(* PLC project SafeLOGIC, BrAutomation SafeDESIGNER  5.24.1.0 *)
(* stored: companyURL http://www.br-automation.com, creationDateTime Fri Nov 28 14:27:25 2025 *)

PROGRAM Main
  VAR  (* added by the conversion: wires and edge detectors of the diagram *)
    _AND_S29_OUT : ANY;
    _AND_S41_OUT : ANY;
  END_VAR

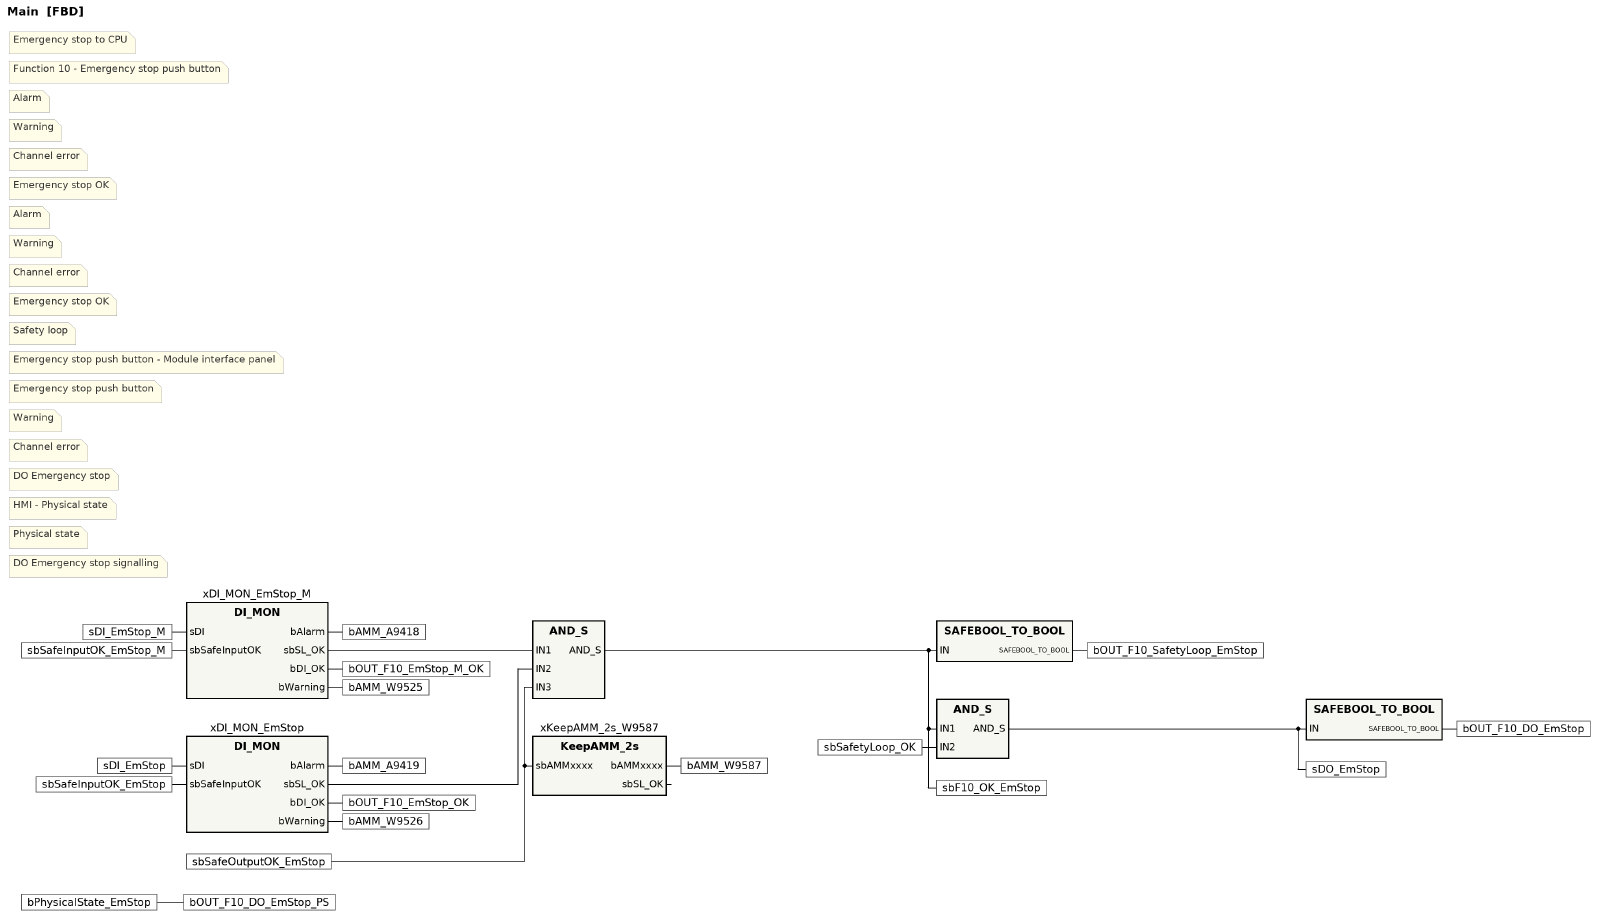
(* FBD diagram, written out as Structured Text *)
(* Function 10 - Emergency stop push button *)
(* Emergency stop push button - Module interface panel *)
(* Alarm *)
xDI_MON_EmStop_M(sDI := sDI_EmStop_M, sbSafeInputOK := sbSafeInputOK_EmStop_M);
bAMM_A9418 := xDI_MON_EmStop_M.bAlarm;
(* Emergency stop OK *)
(* Channel error *)
(* Warning *)
bAMM_W9525 := xDI_MON_EmStop_M.bWarning;
bOUT_F10_EmStop_M_OK := xDI_MON_EmStop_M.bDI_OK;
(* Emergency stop push button *)
(* Alarm *)
xDI_MON_EmStop(sDI := sDI_EmStop, sbSafeInputOK := sbSafeInputOK_EmStop);
bAMM_A9419 := xDI_MON_EmStop.bAlarm;
(* Emergency stop OK *)
(* Channel error *)
(* Warning *)
bAMM_W9526 := xDI_MON_EmStop.bWarning;
bOUT_F10_EmStop_OK := xDI_MON_EmStop.bDI_OK;
(* Safety loop *)
(* Emergency stop to CPU *)
_AND_S29_OUT := AND_S(xDI_MON_EmStop_M.sbSL_OK, xDI_MON_EmStop.sbSL_OK, sbSafeOutputOK_EmStop);
bOUT_F10_SafetyLoop_EmStop := SAFEBOOL_TO_BOOL(_AND_S29_OUT);
sbF10_OK_EmStop := _AND_S29_OUT;
(* DO Emergency stop *)
(* DO Emergency stop signalling *)
_AND_S41_OUT := AND_S(_AND_S29_OUT, sbSafetyLoop_OK);
sDO_EmStop := _AND_S41_OUT;
bOUT_F10_DO_EmStop := SAFEBOOL_TO_BOOL(_AND_S41_OUT);
(* Channel error *)
(* Warning *)
xKeepAMM_2s_W9587(sbAMMxxxx := sbSafeOutputOK_EmStop);
bAMM_W9587 := xKeepAMM_2s_W9587.bAMMxxxx;
(* HMI - Physical state *)
(* Physical state *)
bOUT_F10_DO_EmStop_PS := bPhysicalState_EmStop;
END_PROGRAM
